// TwinCAT 3 PLC project PLC
// ProgramVersion: 3.1.4024.0
// libraries:
//   SPT Base Types, * (Beckhoff Automation LLC)
//   SPT Components, * (Beckhoff Automation LLC)
//   SPT Diagnostic, * (Beckhoff Automation LLC)
//   SPT EtherCat, * (Beckhoff Automation LLC)
//   SPT Event Logger, * (Beckhoff Automation LLC)
//   SPT Kinematics, * (Beckhoff Automation LLC)
//   SPT Motion Control, * (Beckhoff Automation LLC)
//   SPT NCI, * (Beckhoff Automation LLC)
//   SPT Utilities, * (Beckhoff Automation LLC)
//   SPT Vision, * (Beckhoff Automation LLC)
//   SPT XTS, * (Beckhoff Automation LLC)
//   Tc2_MC2, * (Beckhoff Automation GmbH)
//   Tc2_Standard, * (Beckhoff Automation GmbH)
//   Tc2_System, * (Beckhoff Automation GmbH)
//   Tc3_EventLogger, * (Beckhoff Automation GmbH)
//   Tc3_Module, * (Beckhoff Automation GmbH)
//   Tc3_PackML_V2, * (Beckhoff Automation GmbH)
// project tree:
//   / GlobalTextList.TcGTLO, PlcTask.TcTTO (not stored), Visualization Manager.TcVMO (not stored)
//   POUs/ FB_HomeRoutine_CalibrationCam.TcPOU, FB_Machine.TcPOU, MAIN.TcPOU
//   VISUs/ Visualization.TcVIS
// real-time tasks:
//   TASK PlcTask: cycle T#10ms, priority 20, ADS port 350
// motion (NC):
// variable links:
//   PLC/PLC Instance <-> NC-Task 1 SAF/Axes/Axis 1
//     PlcTask Inputs/MAIN.Machine.VAxis.BasicAxis._Axis.NcToPlc <-> Outputs/ToPlc
//     PlcTask Outputs/MAIN.Machine.VAxis.BasicAxis._Axis.PlcToNc <-> Inputs/FromPlc

// ---- POUs/FB_HomeRoutine_CalibrationCam.TcPOU
FUNCTION_BLOCK FB_HomeRoutine_CalibrationCam EXTENDS FB_CyclicFB IMPLEMENTS I_MotionSequence
VAR
	_Axis : I_BasicAxis;

	//
	MCHomeCalCam	: MC_Home;
	_HomingDn		: BOOL;
	SequenceStep	: UDINT;
	_Position		: LREAL;
	_Options		: ST_HomingOptions;
	_CalibrationCam : BOOL;
END_VAR

PROPERTY Axis : I_BasicAxis
GET
Axis := _Axis;
END_GET
SET
_Axis := Axis;
END_SET
END_PROPERTY

PROPERTY CalibrationCam : BOOL
GET
CalibrationCam := _CalibrationCam;
END_GET
SET
_CalibrationCam := CalibrationCam;
END_SET
END_PROPERTY

METHOD PUBLIC CyclicLogic
CASE SequenceStep OF
	10:
		MCHomeCalCam(Axis			 := _Axis.Axis,
					 Execute		 := TRUE,
					 Position		 := _Position,
					 HomingMode		 := MC_HomingMode.MC_DefaultHoming,
					 Options		 := _Options,
					 bCalibrationCam := _CalibrationCam);

		IF NOT MCHomeCalCam.Busy THEN
			IF MCHomeCalCam.Error THEN
				_Error		 := TRUE;
				_ErrorID	 := MCHomeCalCam.ErrorID;
				SequenceStep := 0;
			ELSE
				//No error occurred
				SequenceStep := 0;
			END_IF

			MCHomeCalCam(Axis := _Axis.Axis, Execute := FALSE);
		END_IF
END_CASE

_Busy := SequenceStep <> 0;
END_METHOD

METHOD Execute : BOOL
IF (_Axis = 0) OR _Busy THEN
	RETURN;
END_IF

_Busy		 := TRUE;
_Error		 := FALSE;
_ErrorID	 := 0;
_HomingDn	 := FALSE;
SequenceStep := 10;
Execute		 := TRUE;
END_METHOD

PROPERTY Options : ST_HomingOptions
GET
Options := _Options;
END_GET
SET
_Options := Options;
END_SET
END_PROPERTY

PROPERTY Position : LREAL
GET
Position := _Position;
END_GET
SET
_Position := Position;
END_SET
END_PROPERTY

END_FUNCTION_BLOCK

// ---- POUs/FB_Machine.TcPOU
FUNCTION_BLOCK FB_Machine EXTENDS FB_PackML_BaseModule
VAR
	VAxis	  : FB_Component_BasicAxis := (Name := 'V Axis');
	Home	  : BOOL;
	AxisHomed : BOOL;

	//Home Commands
	HomeAbs		 : BOOL;
	HomeHardStop : BOOL;
	HomeSetPos	 : BOOL;
	HomeCalCam	 : BOOL;

	//Homing Options
	AbsHoming	   : FB_HomeRoutine_AbsHoming;
	HardStopHoming : FB_HomeRoutine_HardStop;
	SetPosition	   : FB_HomeRoutine_SetPosition;
	CalibrationCam : FB_HomeRoutine_CalibrationCam;
END_VAR

//! @summary This method serves as the entry point for all underlying FB logic

//! @description This method should be called cyclically by descendant function blocks by invoking <c>SUPER^.CyclicLogic()</c>.  Alternatively, the contents of this method could be reimplemented entirely in which case a call to this method would not be necessary.
METHOD PUBLIC CyclicLogic
VAR
	i : UDINT;
END_VAR
IF NOT _InitComplete THEN
	_InitComplete := Initialize();
	RETURN;
END_IF

SUPER^.CyclicLogic();
END_METHOD

//! @summary This method contains code which will execute when this PackML module is in the <b>Execute</b> state
METHOD PROTECTED Execute
(*! <description> <b>The base implementation of this method is empty. User must override this method to provide functionality.</b>
<table> 
	<tr>
		<th> Previous State </th>
		<th> Transition In </th>
		<th> Transition Out </th>
		<th> Next State  </th> 
	</tr>
	<tr>
		<td> Starting<b>-or-</b>Unholding <b>-or-</b>Unsuspending</td>
		<td> State Complete<i>(Starting<b>-or-</b>Unholding<b>-or-</b>Unsuspending)</i></td> 
		<td> State Complete<b>-or-</b>Hold Command<b>-or-</b>Suspend Command</td>
		<td> Completing<b>-or-</b>Holding<b>-or-</b>Suspending</td>
	</tr>
</table>
This method is called as required by <c>StateControl()</c>
</description> 

*)
VAR
END_VAR
CASE SequenceState OF
	0:
		IF HomeAbs THEN
			HomeAbs			 := FALSE;
			VAxis.HomeMethod := AbsHoming;
			SequenceState	 := SequenceState + 10;
		END_IF

		IF HomeHardStop THEN
			HomeHardStop	 := FALSE;
			VAxis.HomeMethod := HardStopHoming;
			SequenceState	 := SequenceState + 10;
		END_IF

		IF HomeSetPos THEN
			HomeSetPos		 := FALSE;
			VAxis.HomeMethod := SetPosition;
			SequenceState	 := SequenceState + 10;
		END_IF

		IF HomeCalCam THEN
			HomeCalCam		 := FALSE;
			VAxis.HomeMethod := CalibrationCam;
			SequenceState	 := SequenceState + 10;
		END_IF

	10:
		IF VAxis.Home() THEN
			SequenceState := SequenceState + 10;
		END_IF

	20:
		IF VAxis.Axis.Status.Homed THEN
			SequenceState := SequenceState + 10;
		END_IF

	30:
		AxisHomed := TRUE;
END_CASE
END_METHOD

METHOD hmip
VAR_INPUT
END_VAR
AllowHMIControl(ThisModuleOnly := TRUE);
END_METHOD

// Automatically enables and disables HMI control based on the PackML mode
METHOD PROTECTED HMIPermissions

// This method is called cyclically by CyclicLogic()
AllowHMIControl(ThisModuleOnly := TRUE);
END_METHOD

//! @summary Basic module initialization logic
METHOD PROTECTED Initialize : BOOL;
VAR
	i						 : UDINT;
	varInfo					 : __SYSTEM.VAR_INFO;
	AllSubUnitsInitialized	 : BOOL := TRUE;
	AllComponentsInitialized : BOOL := TRUE;
END_VAR

//! @description This method is called by <c>CyclicLogic()</c> as required
Initialize := FALSE;
CASE DescendantSequenceState OF
	0:
		RegisterComponent(Component := VAxis);
		DescendantSequenceState := DescendantSequenceState + 10;

	10:
		IF SUPER^.Initialize() THEN
			Initialize := TRUE;
		END_IF
END_CASE
END_METHOD

//! @summary This method contains code which will execute when this PackML module is in the <b>Starting</b> state
METHOD PROTECTED Starting
VAR
	i				: UDINT;
	SubModulesReady : BOOL := TRUE;
END_VAR

(*! <description><b></b><table> 
	<tr>
		<th> Previous State </th>
		<th> Transition In </th>
		<th> Transition Out </th>
		<th> Next State  </th> 
	</tr>
	<tr>
		<td> Idle </td>
		<td> Start Command </td> 
		<td> State Complete </td>
		<td> Execute </td> 
	</tr>
</table>
This method is called as required by <c>StateControl()</c>
</description> 

*)
CASE SequenceState OF
	0:
		NoStateTasksToComplete := FALSE;
		SequenceState		   := SequenceState + 10;

	10:
		IF VAxis.Enable() THEN
			SequenceState := SequenceState + 10;
		END_IF

	20:
		IF VAxis.Enabled THEN
			SequenceState := SequenceState + 10;
		END_IF

	30:
		StateTasksComplete := TRUE;
END_CASE

SUPER^.Starting();
END_METHOD

END_FUNCTION_BLOCK

// ---- POUs/MAIN.TcPOU
PROGRAM MAIN
VAR
	Machine : FB_Machine := (Name := 'Machine');
END_VAR

(*All sample code provided by Beckhoff Automation LLC are for illustrative purposes only and are provided “as is” and without any warranties, express or implied. Actual implementations in applications will vary significantly. Beckhoff Automation LLC shall have no liability for, and does not waive any rights in relation to, any code samples that it provides or the use of such code samples for any purpose.*)

(*
	The FB_Component_BasicAxis within the SPT Components library is configured to use a Homing Routine defined in the SPT_MotionControl library.
	FB_HomeRoutine_SetZeroHere, which is an implementation of the MC_SetPosition from the Tc2_MC2 library. 
	The strategy design pattern is used for HomeMethod, ResetMethod, and ExternalSequence. 
	You can change the default homing routine by declaring an instance of a function block that implements the interface I_MotionSequence, 
	and then passing it to the HomeMethod property of your instance of FB_Component_BasicAxis. 
	Within the SPT Motion Control library we provide three other homing options (FB_HomeRoutine_AbsHoming, FB_HomeRoutine_HardStop, FB_HomeRoutine_SetPosition). 
	Further documentation can be found here: https://beckhoff-usa-community.github.io/SPT-Libraries/SPT_MotionControl/functionblocks.html#home-routines
	
	For this sample project an Axis Component is declared within FB_Machine.
	In the Execute method of FB_Machine one of 4 possible home routines can be selected.
	The first 3 are from the SPT Motion Control library, and the fourth is availble in the project.
	
	To use this sample code, toggle resetStateMachine to place the state machine into Production.Execute
	and then toggle one of the four home routines in the execute mehod to start the homing process.
	
*)

//This is for debug only and should be removed
_AppInfo.KeepOutputsOnBP := TRUE;

//
Machine.CyclicLogic();

END_PROGRAM

// ---- VISUs/Visualization.TcVIS
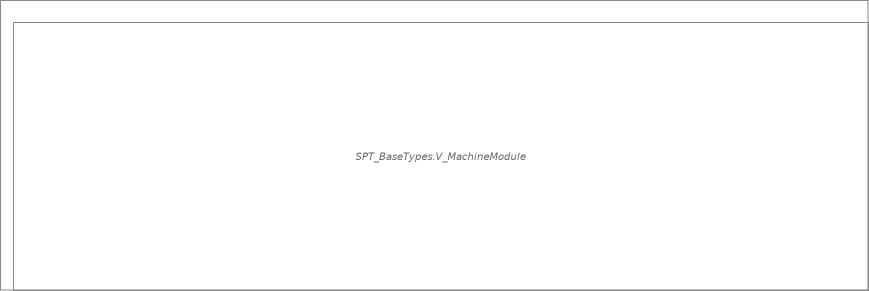
VISUALIZATION Visualization  // 869x291
    Frame (13,22 856x269)
        shows SPT_BaseTypes.V_MachineModule(HMI := MAIN.Machine.PackMLBaseModule_HMI)
END_VISUALIZATION
